RoboDK station: Presenting Piece To The Sewing Machine Triangle.rdk

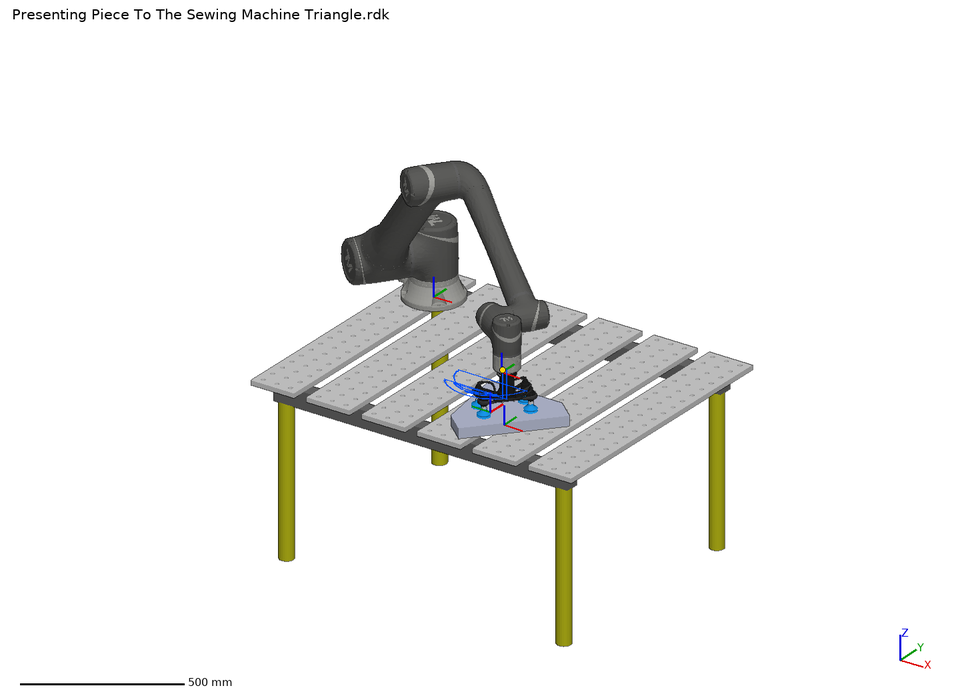
[picture v0: the station drawn from its stored meshes, robots at their saved joint values, targets as dots, program paths as lines]
Station Presenting Piece To The Sewing Machine Triangle (saved by RoboDK 5.1.1). Poses are relative to the parent item; angles as X-Y-Z fixed-axis rotations.
Station parameters (name, value as stored): OPC-UA, opc.tcp://localhost:4840
  - frame Omron TM12X Base at (-555.72, -100.3, 18.7) mm
    - robot Omron TM12X: 6 axes, payload 12 kg, reach 1300 mm, repeatability 0.1 mm, weight 33.3 kg
        modified DH rows (alpha deg, a mm, theta deg, d mm): 0, 0, 0, 165.2; 90, 0, 90, 0; 0, 636.1, 0, 0; 0, 557.9, -90, 156.3; -90, 0, 0, 106; 90, 0, 180, 113.15
        joint limits [-270, -180, -166, -180, -180, -270] to [270, 180, 166, 180, 180, 270]; home [0, 0, 90, 0, 90, 0]; saved at [-34.524, 44.604, 71.291, -25.894, 90, 186.032]
      - tool RobotiQ EPick Four Vacuum Cup, TCP at (0, 24, 144) mm, size 191.2 x 117.6 x 147.9 mm
      - tool Triangle, TCP at (0, 0, 200) mm, size 350 x 299.5 x 35 mm, geometry from Triangle.IGS
      - tool Path1, TCP at (0, 0, 0) mm
  - frame World at (-138.83, -335.01, -27.69) mm
    - object Table at (0, 0, 0) mm, size 1193.8 x 965.2 x 609.6 mm, geometry from Table.sld
    - frame Frame 4 at (175.02, -309.15, 38.15) mm, rotated rx 0 ry 0 rz 90 deg
  - frame Sewing at (109.94, -677.1, 0) mm
  - machining project Triangle1 Settings: rotZ(0) | rotX(0)*rotY(0) | rotz(0) | onStart | onPathStart | onApproach | onPoint | onRetract | onFinish | SetRPM(%1) | SetTool(%1) | Extruder(%1) | default | default | OutOnMov(%1) | OutOffMov(%1) | onPathFinish | M_RunCode(%1)
  - program Triangle1 (76 instructions, listed below)
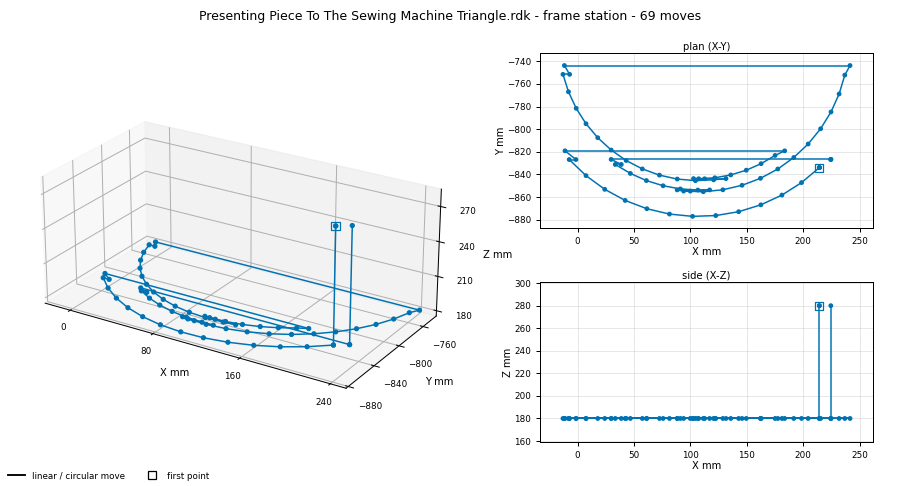
[picture p0: tool path of Presenting Piece To The Sewing Machine Triangle.rdk in frame station, 69 of 69 moves have a stored position in this frame; points joined in program order, loops and branches not executed]

--- program Triangle1 (robot Omron TM12X) ---
  Smooth(1)
  Set speed (1000.0 mm/s)
  Set Ref.: Sewing
  Set Tool: Path1
  Show Path1
  MoveJ 1 to (104.41, -156.91, 280) mm, rotated rx 180 ry 0 rz -134.36 deg; joints [-35.165, 44.394, 71.686, -26.08, 90, -170.806]
  MoveL 2 to (104.41, -156.91, 280) mm, rotated rx 180 ry 0 rz -134.36 deg; joints [-35.165, 44.394, 71.686, -26.08, 90, -170.806]
  MoveL 3 to (104.41, -156.91, 180) mm, rotated rx -180 ry 0 rz -134.36 deg; joints [-35.165, 49.07, 74.374, -33.445, 90, -170.806]
  MoveL 4 to (104.41, -156.91, 180) mm, rotated rx -180 ry 0 rz -134.36 deg; joints [-35.165, 49.07, 74.374, -33.445, 90, -170.806]
  Set speed (50.0 mm/s)
  MoveL 5 to (88.64, -170.14, 180) mm, rotated rx -180 ry 0 rz -141.97 deg; joints [-36.253, 48.905, 74.71, -33.615, 90, -164.286]
  MoveL 6 to (71.25, -181.17, 180) mm, rotated rx -180 ry 0 rz -149.57 deg; joints [-37.305, 48.56, 75.41, -33.971, 90, -157.732]
  MoveL 7 to (52.56, -189.8, 180) mm, rotated rx -180 ry 0 rz -157.18 deg; joints [-38.309, 48.043, 76.46, -34.504, 90, -151.13]
  MoveL 8 to (32.89, -195.87, 180) mm, rotated rx -180 ry 0 rz -164.79 deg; joints [-39.254, 47.365, 77.836, -35.201, 90, -144.468]
  MoveL 9 to (12.59, -199.29, 180) mm, rotated rx -180 ry 0 rz -172.39 deg; joints [-40.127, 46.539, 79.508, -36.047, 90, -137.734]
  MoveL 10 to (-7.98, -200, 180) mm, rotated rx -180 ry 0 rz -180 deg; joints [-40.914, 45.582, 81.443, -37.025, 90, -130.914]
  MoveL 11 to (-28.47, -197.97, 180) mm, rotated rx 180 ry 0 rz 172.39 deg; joints [-41.602, 44.512, 83.602, -38.114, 90, -123.995]
  MoveL 12 to (-48.51, -193.25, 180) mm, rotated rx -180 ry 0 rz 164.79 deg; joints [-42.177, 43.347, 85.947, -39.295, 90, -116.963]
  MoveL 13 to (-67.75, -185.92, 180) mm, rotated rx -180 ry 0 rz 157.18 deg; joints [-42.625, 42.108, 88.438, -40.545, 90, -109.805]
  MoveL 14 to (-85.84, -176.1, 180) mm, rotated rx -180 ry 0 rz 149.57 deg; joints [-42.933, 40.812, 91.032, -41.845, 90, -102.506]
  MoveL 15 to (-102.48, -163.98, 180) mm, rotated rx -180 ry 0 rz 141.97 deg; joints [-43.087, 39.482, 93.689, -43.171, 90, -95.053]
  MoveL 16 to (-117.37, -149.76, 180) mm, rotated rx -180 ry 0 rz 134.36 deg; joints [-43.073, 38.137, 96.367, -44.504, 90, -87.432]
  MoveL 17 to (-111.4, -149.76, 180) mm, rotated rx -180 ry 0 rz 134.36 deg; joints [-42.814, 38.374, 95.895, -44.27, 90, -87.173]
  MoveL 18 to (-121.09, -142.04, 180) mm, rotated rx -180 ry 0 rz 130.56 deg; joints [-42.873, 37.588, 97.458, -45.045, 90, -83.429]
  MoveL 19 to (73.67, -142.04, 180) mm, rotated rx -180 ry 0 rz 130.56 deg; joints [-35.477, 46.575, 79.435, -36.01, 90, -76.033]
  MoveL 20 to (65.16, -146.14, 180) mm, rotated rx -180 ry 0 rz 127.18 deg; joints [-35.944, 46.335, 79.92, -36.255, 90, -73.12]
  MoveL 21 to (52.78, -153.42, 180) mm, rotated rx -180 ry 0 rz 120.42 deg; joints [-36.69, 46.068, 80.461, -36.529, 90, -67.106]
  MoveL 22 to (39.62, -159.19, 180) mm, rotated rx 180 ry 0 rz 113.66 deg; joints [-37.4, 45.696, 81.212, -36.908, 90, -61.058]
  MoveL 23 to (25.88, -163.37, 180) mm, rotated rx -180 ry 0 rz 106.9 deg; joints [-38.069, 45.226, 82.163, -37.388, 90, -54.967]
  MoveL 24 to (11.74, -165.9, 180) mm, rotated rx 180 ry 0 rz 100.14 deg; joints [-38.688, 44.663, 83.297, -37.96, 90, -48.827]
  MoveL 25 to (-2.6, -166.76, 180) mm, rotated rx -180 ry 0 rz 93.38 deg; joints [-39.249, 44.018, 84.598, -38.616, 90, -42.629]
  MoveL 26 to (2.71, -166.76, 180) mm, rotated rx 180 ry 0 rz 93.38 deg; joints [-39.054, 44.272, 84.087, -38.358, 90, -42.434]
  MoveL 27 to (-7.13, -166.63, 180) mm, rotated rx -180 ry 0 rz 90 deg; joints [-39.411, 43.796, 85.045, -38.841, 90, -39.411]
  MoveL 28 to (21.63, -166.63, 180) mm, rotated rx 180 ry 0 rz 90 deg; joints [-38.366, 45.188, 82.238, -37.426, 90, -38.366]
  MoveL 29 to (10.68, -167.68, 180) mm, rotated rx 180 ry 0 rz 86.25 deg; joints [-38.806, 44.707, 83.209, -37.916, 90, -35.056]
  MoveL 30 to (-5.46, -168.41, 180) mm, rotated rx -180 ry 0 rz 78.75 deg; joints [-39.429, 43.97, 84.694, -38.664, 90, -28.179]
  MoveL 31 to (-21.56, -167.03, 180) mm, rotated rx 180 ry 0 rz 71.25 deg; joints [-39.97, 43.143, 86.359, -39.501, 90, -21.22]
  MoveL 32 to (-37.34, -163.55, 180) mm, rotated rx 180 ry 0 rz 63.75 deg; joints [-40.417, 42.239, 88.174, -40.413, 90, -14.167]
  MoveL 33 to (-52.53, -158.05, 180) mm, rotated rx 180 ry 0 rz 56.25 deg; joints [-40.76, 41.273, 90.11, -41.383, 90, -7.011]
  MoveL 34 to (-66.88, -150.61, 180) mm, rotated rx 180 ry 0 rz 48.75 deg; joints [-40.99, 40.261, 92.134, -42.395, 90, 0.26]
  MoveL 35 to (-80.13, -141.36, 180) mm, rotated rx 180 ry 0 rz 41.25 deg; joints [-41.098, 39.219, 94.213, -43.432, 90, 7.652]
  MoveL 36 to (-92.06, -130.46, 180) mm, rotated rx 180 ry 0 rz 33.75 deg; joints [-41.074, 38.163, 96.315, -44.478, 90, 15.176]
  MoveL 37 to (-102.46, -118.09, 180) mm, rotated rx -180 ry 0 rz 26.25 deg; joints [-40.912, 37.109, 98.406, -45.516, 90, 22.838]
  MoveL 38 to (-111.16, -104.48, 180) mm, rotated rx 180 ry 0 rz 18.75 deg; joints [-40.608, 36.075, 100.453, -46.528, 90, 30.642]
  MoveL 39 to (-118.01, -89.84, 180) mm, rotated rx 180 ry 0 rz 11.25 deg; joints [-40.159, 35.077, 102.421, -47.499, 90, 38.591]
  MoveL 40 to (-122.89, -74.44, 180) mm, rotated rx 180 ry 0 rz 3.75 deg; joints [-39.567, 34.133, 104.279, -48.412, 90, 46.683]
  MoveL 41 to (-117.01, -74.44, 180) mm, rotated rx 180 ry 0 rz 3.75 deg; joints [-39.31, 34.37, 103.812, -48.183, 90, 46.94]
  MoveL 42 to (-121.63, -66.63, 180) mm, rotated rx 180 ry 0 rz 0 deg; joints [-39.095, 33.809, 104.915, -48.724, 90, 50.905]
  MoveL 43 to (131.63, -66.63, 180) mm, rotated rx 180 ry 0 rz 0 deg; joints [-30.129, 46.079, 80.439, -36.518, 90, 59.871]
  MoveL 44 to (126.99, -75.09, 180) mm, rotated rx 180 ry 0 rz -3.75 deg; joints [-30.675, 46.209, 80.176, -36.385, 90, 63.075]
  MoveL 45 to (121.94, -91.79, 180) mm, rotated rx 180 ry 0 rz -11.25 deg; joints [-31.627, 46.72, 79.142, -35.862, 90, 69.623]
  MoveL 46 to (114.75, -107.69, 180) mm, rotated rx 180 ry 0 rz -18.75 deg; joints [-32.594, 47.093, 78.386, -35.479, 90, 76.156]
  MoveL 47 to (105.54, -122.52, 180) mm, rotated rx 180 ry 0 rz -26.25 deg; joints [-33.567, 47.321, 77.925, -35.246, 90, 82.683]
  MoveL 48 to (94.49, -136.01, 180) mm, rotated rx 180 ry 0 rz -33.75 deg; joints [-34.533, 47.399, 77.767, -35.166, 90, 89.217]
  MoveL 49 to (81.76, -147.95, 180) mm, rotated rx 180 ry 0 rz -41.25 deg; joints [-35.484, 47.325, 77.917, -35.242, 90, 95.766]
  MoveL 50 to (67.58, -158.13, 180) mm, rotated rx 180 ry 0 rz -48.75 deg; joints [-36.407, 47.1, 78.371, -35.472, 90, 102.343]
  MoveL 51 to (52.2, -166.36, 180) mm, rotated rx 180 ry 0 rz -56.25 deg; joints [-37.292, 46.731, 79.12, -35.851, 90, 108.958]
  MoveL 52 to (35.88, -172.52, 180) mm, rotated rx 180 ry 0 rz -63.75 deg; joints [-38.128, 46.223, 80.148, -36.371, 90, 115.622]
  MoveL 53 to (18.89, -176.5, 180) mm, rotated rx -180 ry 0 rz -71.25 deg; joints [-38.905, 45.586, 81.434, -37.021, 90, 122.346]
  MoveL 54 to (1.53, -178.22, 180) mm, rotated rx -180 ry 0 rz -78.75 deg; joints [-39.61, 44.833, 82.955, -37.788, 90, 129.14]
  MoveL 55 to (-15.91, -177.66, 180) mm, rotated rx 180 ry 0 rz -86.25 deg; joints [-40.233, 43.977, 84.681, -38.658, 90, 136.017]
  MoveL 56 to (-10.03, -177.66, 180) mm, rotated rx -180 ry 0 rz -86.25 deg; joints [-40.013, 44.253, 84.125, -38.377, 90, 136.237]
  MoveL 57 to (-21.63, -176.63, 180) mm, rotated rx -180 ry 0 rz -90 deg; joints [-40.403, 43.655, 85.328, -38.983, 90, 139.597]
  MoveL 58 to (7.13, -176.63, 180) mm, rotated rx 180 ry 0 rz -90 deg; joints [-39.335, 45.017, 82.584, -37.601, 90, 140.665]
  MoveL 59 to (-3.3, -176.74, 180) mm, rotated rx -180 ry 0 rz -93.38 deg; joints [-39.722, 44.522, 83.582, -38.104, 90, 143.658]
  MoveL 60 to (-18.81, -175.75, 180) mm, rotated rx -180 ry 0 rz -100.14 deg; joints [-40.257, 43.738, 85.161, -38.899, 90, 149.882]
  MoveL 61 to (-34.09, -172.94, 180) mm, rotated rx -180 ry 0 rz -106.9 deg; joints [-40.715, 42.886, 86.875, -39.761, 90, 156.183]
  MoveL 62 to (-48.94, -168.35, 180) mm, rotated rx -180 ry 0 rz -113.66 deg; joints [-41.088, 41.977, 88.7, -40.677, 90, 162.57]
  MoveL 63 to (-63.15, -162.04, 180) mm, rotated rx -180 ry 0 rz -120.42 deg; joints [-41.367, 41.022, 90.613, -41.635, 90, 169.049]
  MoveL 64 to (-76.51, -154.11, 180) mm, rotated rx -180 ry 0 rz -127.18 deg; joints [-41.546, 40.034, 92.588, -42.622, 90, 175.631]
  MoveL 65 to (-71.21, -154.11, 180) mm, rotated rx -180 ry 0 rz -127.18 deg; joints [-41.329, 40.259, 92.138, -42.397, 90, 175.848]
  MoveL 66 to (-80.17, -149.64, 180) mm, rotated rx -180 ry 0 rz -130.56 deg; joints [-41.488, 39.647, 93.361, -43.007, 90, 179.067]
  MoveL 67 to (114.59, -149.64, 180) mm, rotated rx -180 ry 0 rz -130.56 deg; joints [-34.524, 49.262, 73.985, -33.247, 90, 186.032]
  Set speed (1000.0 mm/s)
  MoveL 68 to (114.59, -149.64, 180) mm, rotated rx -180 ry 0 rz -130.56 deg; joints [-34.524, 49.262, 73.985, -33.247, 90, 186.032]
  MoveL 69 to (114.59, -149.64, 280) mm, rotated rx -180 ry 0 rz -130.56 deg; joints [-34.524, 44.604, 71.291, -25.894, 90, 186.032]
